SUBAPPLICATION AX_ASRT_RF_TRIG (* Boolean falling and rising edge detection, gebuendelt als ASRT (SET/RESET, TOGGLE ungenutzt) - aus AX_ASR_RF_TRIG + ASRT_SR_AE_TO_SRT *)
  (* Standard: 61499-2; Description: Copyright (c) 2026 Meisterschulen am Ostbahnhof This program and the accompanying materials are made available under the terms of the Eclipse Public License 2.0 which is available at https://www.eclipse.org/legal/epl-2.0/ SPDX-License-Identifier: EPL-2.0 *)
  (* Version 1.0, 2026-09-06, Franz Höpfinger, Meisterschulen am Ostbahnhof, initial API and implementation and/or initial documentation *)
  PACKAGE MyLib::sys;
  (* Documentation:
  Flankenerkennung, gebündelt als ASRT (SET/RESET)
   Composite statt neuem Low-Level-FBType: wiederverwendet den bestehenden AX_ASR_RF_TRIG (liefert ASR aus einer Flanke) und speist dessen Ausgang direkt in ASRT_SR_AE_TO_SRT (SR_IN) - genau dafür gebaut, ein ASR mit einem optionalen AE-Toggle-Event zu einem ASRT zu kombinieren.
   Funktionsbeschreibung
    - AX_ASR_RF_TRIG_1: steigende Flanke an QI → SET, fallende Flanke → RESET, als gebündeltes ASR.
   - ASRT_SR_AE_TO_SRT_1 übernimmt dieses ASR direkt als SR_IN und bündelt es zu ASRT_OUT. Der zweite Socket (TOGGLE_IN, ein einzelnes AE-Event) bleibt hier unverdrahtet und feuert nie, weil sich aus einem reinen Flankensignal kein unabhängiges drittes Ereignis ableiten lässt.
    Verwendet z.B. in Uebung_232_AX als eine von zwei ASRT-Quellen für ASRT_MERGE_2.
  *)
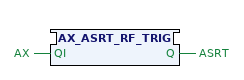
  SOCKETS
    QI : adapter::types::unidirectional::AX; (* value to check for a rising or falling edge *)
  END_SOCKETS
  PLUGS
    Q : adapter::types::unidirectional::ASRT; (* Set/Reset Output (Toggle wird nie gefeuert) *)
  END_PLUGS
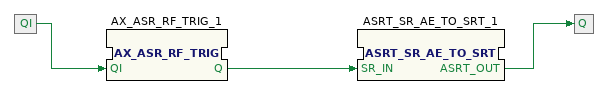
  FBS
    AX_ASR_RF_TRIG_1 : adapter::events::unidirectional::AX_ASR_RF_TRIG;
    ASRT_SR_AE_TO_SRT_1 : adapter::conversion::unidirectional::ASRT_SR_AE_TO_SRT;
  END_FBS
  ADAPTER_CONNECTIONS
    QI TO AX_ASR_RF_TRIG_1.QI;
    AX_ASR_RF_TRIG_1.Q TO ASRT_SR_AE_TO_SRT_1.SR_IN;
    ASRT_SR_AE_TO_SRT_1.ASRT_OUT TO Q;
  END_CONNECTIONS
END_SUBAPPLICATION
